# EPICS substitutions: lsredis/iocBoot/iocCygwin/asynRecord.substitutions
file "$(ASYN)/db/asynRecord.db"
{
pattern
{P        R         PORT    ADDR    OMAX  IMAX}
{lsredis:     asyn_1   serial1    0     256  256}
{lsredis:     asyn_2   serial2    0     256  256}
{lsredis:     asyn_3   serial3    0     256  256}
{lsredis:     asyn_4   serial4    0     256  256}
}
